Staubli VAL3: page.pjx

Parameters version=s7.1 stackSize=50000 millimeterUnit=true
Program file=main.pgx
Data file=page.dtx
